// TIA Portal project "modbus_slave" (V15.1)

(* hardware
DEVICE "S7-1200 station_1"  S7-1200 Station
   slot 0: "Rack_0"  S7-1200 Rack  Rack  V1.0
   slot 1: "PLC_1"  CPU 1214C DC/DC/DC  6ES7 214-1AG40-0XB0  V4.2
*)

// ===== PLC "PLC_1"  CPU 1214C DC/DC/DC =====

VAR_GLOBAL   // PLC tag table "默认变量表"
   "System_Byte" AT %MB1 : Byte;
   "FirstScan" AT %M1.0 : Bool;
   "DiagStatusUpdate" AT %M1.1 : Bool;
   "AlwaysTRUE" AT %M1.2 : Bool;
   "AlwaysFALSE" AT %M1.3 : Bool;
   "Clock_Byte" AT %MB0 : Byte;
   "Clock_10Hz" AT %M0.0 : Bool;
   "Clock_5Hz" AT %M0.1 : Bool;
   "Clock_2.5Hz" AT %M0.2 : Bool;
   "Clock_2Hz" AT %M0.3 : Bool;
   "Clock_1.25Hz" AT %M0.4 : Bool;
   "Clock_1Hz" AT %M0.5 : Bool;
   "Clock_0.625Hz" AT %M0.6 : Bool;
   "Clock_0.5Hz" AT %M0.7 : Bool;
   "Tag_1" AT %I0.0 : Bool;
   "Rw_NDR" AT %M2.0 : Bool;
   "Rw_DR" AT %M2.1 : Bool;
   "Rw_ERROR" AT %M2.2 : Bool;
   "Rf_NDR" AT %M2.3 : Bool;
   "Rf_DR" AT %M2.4 : Bool;
   "Rf_ERROR" AT %M2.5 : Bool;
   "Rdi_NDR" AT %M2.6 : Bool;
   "Rdi_DR" AT %M2.7 : Bool;
   "Rdi_ERROR" AT %M3.0 : Bool;
   "Rdo_NDR" AT %M3.1 : Bool;
   "Rdo_DR" AT %M3.2 : Bool;
   "Rdo_ERROR" AT %M3.3 : Bool;
   "Rw_STATUS" AT %MW4 : Word;
   "Rw_ERRORCODE" AT %MW6 : Word;
   "Rf_STATUS" AT %MW8 : Word;
   "Rf_ERRORCODE" AT %MW10 : Word;
   "Rdi_STATUS" AT %MW12 : Word;
   "Rdi_ERRORCODE" AT %MW14 : Word;
   "Rdo_STATUS" AT %MW16 : Word;
   "Rdo_ERRORCODE" AT %MW18 : Word;
   "Tag_2" AT %IW64 : Word;
   "Tag_3" AT %IW66 : Word;
END_VAR

DATA_BLOCK "Net_Info"   // DB2
{ S7_Optimized_Access := 'TRUE' }
VERSION : 0.1
   VAR
      modbus_rt : TCON_IP_v4;
   END_VAR
BEGIN
   modbus_rt.InterfaceId := 64;
   modbus_rt.ID := 1;
   modbus_rt.ConnectionType := 11;
   modbus_rt.ActiveEstablished := 0;
   modbus_rt.LocalPort := 502;
END_DATA_BLOCK

DATA_BLOCK "Data_Modbus"   // DB3
{ S7_Optimized_Access := 'FALSE' }
VERSION : 0.1
   VAR
      float_reg : Array[0..1] of Real;
      word_reg : Array[0..32] of Word;
      di_reg : Array[0..32] of Bool;
      do_reg : Array[0..32] of Bool;
   END_VAR
BEGIN
END_DATA_BLOCK

ORGANIZATION_BLOCK "Main"   // OB1, LAD, ProgramCycle
TITLE = "Main Program Sweep (Cycle)"
{ S7_Optimized_Access := 'TRUE' }
VERSION : 0.1
   VAR_INPUT
      Initial_Call : Bool;   // Initial call of this OB
      Remanence : Bool;   // =True, if remanent data are available
   END_VAR
BEGIN

REGION Network 1: Modbus Slave
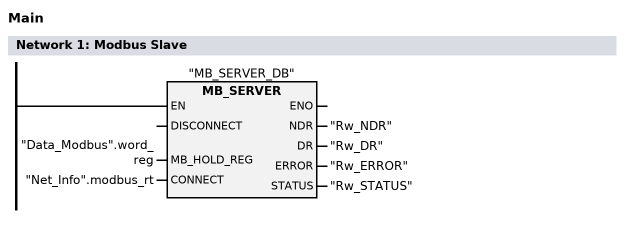
   "MB_SERVER_DB"(MB_HOLD_REG := "Data_Modbus".word_reg,   // MB_SERVER
                  CONNECT := "Net_Info".modbus_rt,
                  NDR => "Rw_NDR",
                  DR => "Rw_DR",
                  ERROR => "Rw_ERROR",
                  STATUS => "Rw_STATUS");
END_REGION
END_ORGANIZATION_BLOCK